# EPICS autosave request: iocBoot/iocInjEfficiency/auto_settings_injEfficiency.req
file "injEfficiency_settings.req",                P=$(P),  R=$(R)
